ABB RobotStudio station: miniproject_v1_20180423-160942.rsstn

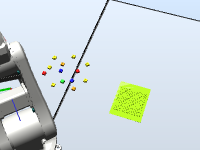
Station Station (saved by RobotStudio 6.6.7701.1025)
Controller miniproject
  mechanical unit ROB_1: IRB120_3_58__01, 6 joints, base frame (0, 0, 0) mm
Layout (positions relative to the parent item):
  - IRB120_3_58__01 [mechanism, from Robots\IRB120_3_58_G_01.rslib] at (0, 0, 0) mm; joint values [0.7906, 0.5123, 0.4141, -0.1232, 0.6528, 0.3656] (rad or m)
  - Deliver plate 16x16 LEGO Plate [part] at (400, -300, 0) mm
  - lego2x2 Orange [part] at (372.6, -24.86, 0) mm, rotated rx 90 ry 0 rz 0 deg
  - lego2x2 Yellow [part] at (549.33, 43.86, 0) mm, rotated rx 90 ry 0 rz 0 deg
  - lego2x2 Blue [part] at (414.35, 0.66, 0) mm, rotated rx 90 ry 0 rz -26 deg
  - lego2x2 Blue_4 [part] at (448.59, 72, 0) mm, rotated rx 90 ry 0 rz 0 deg
  - lego2x2 Green_4 [part] at (395.13, 41.77, 0) mm, rotated rx 90 ry 0 rz -16 deg
  - lego2x2 Orange_4 [part] at (488.39, 78.35, 0) mm, rotated rx 90 ry 0 rz 0 deg
  - lego2x2 Yellow [part] at (450.89, 132.39, 0) mm, rotated rx 90 ry 0 rz -7 deg
  - lego2x2 Yellow_2 [part] at (433.91, -61.74, 0) mm, rotated rx 90 ry 0 rz 0 deg
  - lego2x2 Yellow_3 [part] at (513.14, 132.44, 0) mm, rotated rx 90 ry 0 rz -10 deg
  - lego2x2 Yellow_4 [part] at (361.28, 75.07, 0) mm, rotated rx 90 ry 0 rz 0 deg
  - lego2x2 Yellow_5 [part] at (525.36, -42.12, 0) mm, rotated rx 90 ry 0 rz 50 deg
  - lego2x2 Red_3 [part] at (408.9, 142.68, 0) mm, rotated rx 90 ry 0 rz 0 deg
  - lego2x2 Red_4 [part] at (471.54, -9.93, 0) mm, rotated rx 90 ry 0 rz 35 deg
  - SmartComponent_1 [smart component, from Libraries\SCHINK_WSG_GRIPPER.rslib] at (263.66, 258.76, 254.16) mm, rotated rx -175.8 ry 0.87 rz -149.99 deg
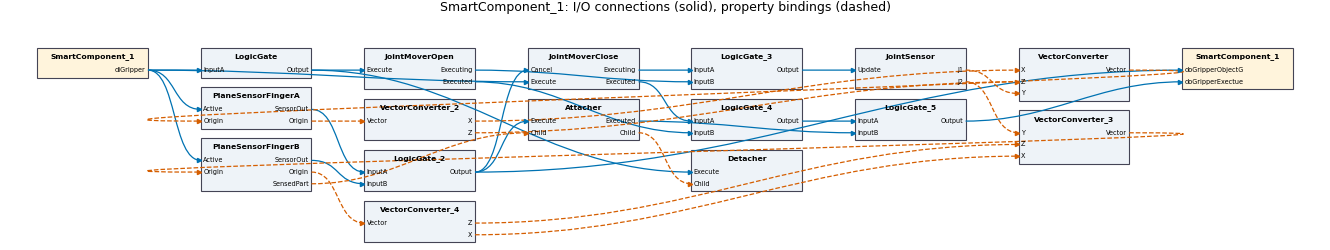
      connections:
        SmartComponent_1.diGripper -> LogicGate.InputA
        SmartComponent_1.diGripper -> PlaneSensorFingerA.Active
        SmartComponent_1.diGripper -> PlaneSensorFingerB.Active
        PlaneSensorFingerA.SensorOut -> LogicGate_2.InputA
        PlaneSensorFingerB.SensorOut -> LogicGate_2.InputB
        LogicGate_2.Output -> JointMoverClose.Cancel
        LogicGate_2.Output -> SmartComponent_1.doGripperObjectGrasped
        SmartComponent_1.diGripper -> JointMoverClose.Execute
        LogicGate.Output -> JointMoverOpen.Execute
        JointMoverClose.Executing -> LogicGate_3.InputA
        JointMoverOpen.Executing -> LogicGate_3.InputB
        LogicGate_3.Output -> JointSensor.Update
        LogicGate_2.Output -> Attacher.Execute
        LogicGate.Output -> Detacher.Execute
        JointMoverClose.Executed -> LogicGate_4.InputA
        JointMoverOpen.Executed -> LogicGate_4.InputB
        LogicGate_4.Output -> LogicGate_5.InputA
        Attacher.Executed -> LogicGate_5.InputB
        LogicGate_5.Output -> SmartComponent_1.doGripperExectued
        VectorConverter_2.X => VectorConverter.X
        VectorConverter_2.Z => VectorConverter.Z
        JointSensor.J1 => VectorConverter.Y
        PlaneSensorFingerA.Origin => VectorConverter_2.Vector
        VectorConverter.Vector => PlaneSensorFingerA.Origin
        JointSensor.J2 => VectorConverter_3.Y
        VectorConverter_4.Z => VectorConverter_3.Z
        VectorConverter_4.X => VectorConverter_3.X
        PlaneSensorFingerB.Origin => VectorConverter_4.Vector
        VectorConverter_3.Vector => PlaneSensorFingerB.Origin
        PlaneSensorFingerB.SensedPart => Attacher.Child
        Attacher.Child => Detacher.Child
    - SCHINK_WSG_GRIPPER [mechanism, from Libraries\SCHINK_WSG_GRIPPER.rslib] at (0, 0, 0) mm; joint values [0.0535, -0.0535] (rad or m)
    - PlaneSensorFingerA [smart component, from Components\PlaneSensor.rslib]
        properties: Origin=[-0.015 0.0535 0.13582]; Axis1=[0.03 0 0]; Axis2=[0 0 0.099]; SensedPart=(none)
      - _sensorPart_ [part]
    - PlaneSensorFingerB [smart component, from Components\PlaneSensor.rslib]
        properties: Origin=[-0.015 -0.0535 0.13582]; Axis1=[0.03 0 0]; Axis2=[0 0 0.099]; SensedPart=(none)
      - _sensorPart_ [part]
    - JointMoverClose [smart component, from Components\JointMover.rslib]
        properties: Mechanism=SCHINK_WSG_GRIPPER; Relative=false; Duration=2; J1=0; J2=0
    - JointMoverOpen [smart component, from Components\JointMover.rslib]
        properties: Mechanism=SCHINK_WSG_GRIPPER; Relative=false; Duration=2; J1=0.0535; J2=-0.0535
    - LogicGate [smart component, from Components\LogicGate.rslib]
        properties: Operator=NOT; Delay=0
    - LogicGate_2 [smart component, from Components\LogicGate.rslib]
        properties: Operator=AND; Delay=0
    - JointSensor [smart component, from Components\JointSensor.rslib]
        properties: Mechanism=SCHINK_WSG_GRIPPER; J1=0.0535; J2=-0.0535
    - LogicGate_3 [smart component, from Components\LogicGate.rslib]
        properties: Operator=OR; Delay=0
    - VectorConverter [smart component, from Components\VectorConverter.rslib]
        properties: X=-0.015; Y=0.0535; Z=0.13582; Vector=[-0.015 0.0535 0.13582]
    - VectorConverter_2 [smart component, from Components\VectorConverter.rslib]
        properties: X=-0.015; Y=0.0535; Z=0.13582; Vector=[-0.015 0.0535 0.13582]
    - VectorConverter_3 [smart component, from Components\VectorConverter.rslib]
        properties: X=-0.015; Y=-0.0535; Z=0.13582; Vector=[-0.015 -0.0535 0.13582]
    - VectorConverter_4 [smart component, from Components\VectorConverter.rslib]
        properties: X=-0.015; Y=-0.0535; Z=0.13582; Vector=[-0.015 -0.0535 0.13582]
    - Attacher [smart component, from Components\Attacher.rslib]
        properties: Parent=SCHINK_WSG_GRIPPER; Flange=0; Child=(none); Mount=false; Offset=[0 0 0]; Orientation=[0 0 0]
    - Detacher [smart component, from Components\Detacher.rslib]
        properties: Child=(none); KeepPosition=true
    - LogicGate_4 [smart component, from Components\LogicGate.rslib]
        properties: Operator=OR; Delay=0
    - LogicGate_5 [smart component, from Components\LogicGate.rslib]
        properties: Operator=OR; Delay=0
  - MoveToViewpoint [smart component, from Components\MoveToViewpoint.rslib] at (262.91, 31.88, 0) mm
      properties: Viewpoint=Viewpoint_7; Time=0
  - Camera [smart component, from Components\Camera.rslib]
      properties: Path=D:\2. P8 Project\Courses\Miniprojects\RV\Simulation\Matlab_simulation_brickstacker; File Name=withBlocks
Attachment: SmartComponent_1 is attached to IRB120_3_58__01 / Link6
Attachment: MoveToViewpoint is attached to lego2x2 Yellow_5
Station signals: DI diGripper, DO doGripperExectued
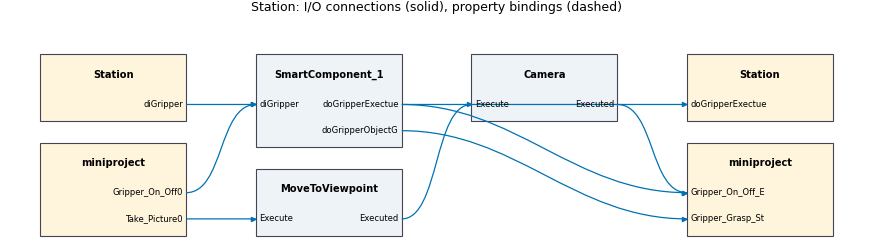
Station logic (signal -> signal, property => property):
  Station.diGripper -> SmartComponent_1.diGripper
  SmartComponent_1.doGripperExectued -> Station.doGripperExectued
  miniproject.Gripper_On_Off0 -> SmartComponent_1.diGripper
  SmartComponent_1.doGripperExectued -> miniproject.Gripper_On_Off_Executed0
  SmartComponent_1.doGripperObjectGrasped -> miniproject.Gripper_Grasp_State0
  MoveToViewpoint.Executed -> Camera.Execute
  miniproject.Take_Picture0 -> MoveToViewpoint.Execute
  Camera.Executed -> miniproject.Gripper_On_Off_Executed0
Targets, tools, work objects and paths stored in the station, written as RAPID:
! task T_ROB1
MODULE FunctionHandler
  PERS tooldata defaultTool:=[TRUE,[[0,0,0],[1,0,0,0]],[1,[0,0,0.001],[1,0,0,0],0,0,0]];
  PERS wobjdata defaultWobj:=[FALSE,TRUE,"",[[0,0,0],[1,0,0,0]],[[0,0,0],[1,0,0,0]]];
  VAR signaldo defaultTakePictureActivationIO;
  VAR signaldi defaultTakePictureExecutedIO;
  PROC FH_TakePicture()
    SetDO defaultTakePictureActivationIO,1;
    WaitDI defaultTakePictureExecutedIO,1;
    SetDO defaultTakePictureActivationIO,0;
  ENDPROC
ENDMODULE

! task T_ROB1
MODULE CommandHandler
  PROC COMH_CommandListener()
  ENDPROC
ENDMODULE

! task T_ROB1
MODULE Module1
  PROC main()
    IP_Initialize;
    COMH_CommandListener;
  ENDPROC
ENDMODULE

! task T_ROB1
MODULE InitParameters
  PROC IP_Initialize()
    ConfL \Off;
    ConfJ \Off;
  ENDPROC
ENDMODULE

! task T_ROB1
MODULE CalibData
  PERS tooldata SCHINK_WSG_GRIPPER_TOOL:=[TRUE,[[0,0,234.82],[1,0,0,0]],[5,[0,0,100],[1,0,0,0],0,0,0]];
ENDMODULE

